// TIA Portal V20 export
TYPE "typeEmHomedCheck"
// stored: Access Published, Namespace Unit1.Em1
   STRUCT
      cmUnWinderAxisB : Bool;
      cmAirShaftOnOff : Bool;
      cmExpelFwdBwd : Bool;
      cmEpc : Bool;
      cmSyncNode : Bool;
   END_STRUCT;
END_TYPE
